FUNCTION_BLOCK DO_2ACTION (* Basic Function Block Type *)
  (* Standard: 61499-2 *)
  (* Version 0.0, 2/8/2023, brink, Flexbridge AB, Template *)
  PACKAGE UAO.Hackathon;
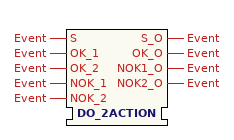
  EVENT_INPUT
    S; (* Action start *)
    OK_1; (* Action done *)
    OK_2;
    NOK_1;
    NOK_2;
  END_EVENT
  EVENT_OUTPUT
    S_O;
    OK_O;
    NOK1_O;
    NOK2_O;
  END_EVENT
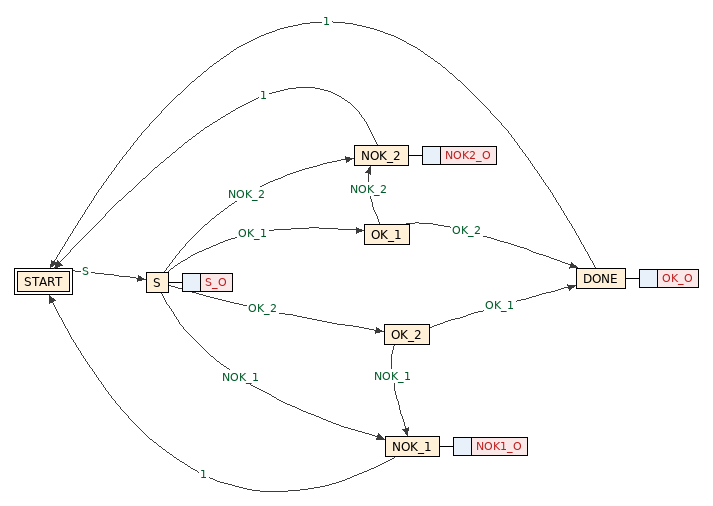
  EC_STATES
    START; (* Initial State *)
    S : -> S_O;
    OK_1;
    NOK_1 : -> NOK1_O;
    DONE : -> OK_O;
    OK_2;
    NOK_2 : -> NOK2_O;
  END_STATES
  EC_TRANSITIONS
    START TO S := S;
    S TO NOK_1 := NOK_1;
    NOK_1 TO START := 1;
    S TO OK_1 := OK_1;
    DONE TO START := 1;
    OK_1 TO DONE := OK_2;
    S TO OK_2 := OK_2;
    OK_2 TO DONE := OK_1;
    OK_2 TO NOK_1 := NOK_1;
    S TO NOK_2 := NOK_2;
    OK_1 TO NOK_2 := NOK_2;
    NOK_2 TO START := 1;
  END_TRANSITIONS
END_FUNCTION_BLOCK
